// set alarm class
SIf.Alm[1].eAlmClass := E_AlmClass.EOFF;
SIf.Alm[1].strText := 'Communication Error to Line Controller'; 
SIf.Alm[2].eAlmClass := E_AlmClass.EOFF;
SIf.Alm[2].strText := 'Emergency Button pressed';
SIf.Alm[3].eAlmClass := E_AlmClass.INFO;
SIf.Alm[3].strText := 'Communication Error to Line Controller'; 
SIf.Alm[4].eAlmClass := E_AlmClass.INFO;
SIf.Alm[4].strText := 'Line to charge already busy, Job not possible';
SIf.Alm[5].eAlmClass := E_AlmClass.INFO;
SIf.Alm[5].strText := 'False Job Parameter';
SIf.Alm[6].eAlmClass := E_AlmClass.INFO;
SIf.Alm[6].strText := 'Hashtable full, no more input possible';
SIf.Alm[7].eAlmClass := E_AlmClass.INFO;
SIf.Alm[7].strText := 'Data Channel Error Receive Data';
SIf.Alm[8].eAlmClass := E_AlmClass.INFO;
SIf.Alm[8].strText := 'Data Channel Error Send Data';

//*******************************************************************************
// initial values
//*******************************************************************************
// software configuration
CIf.SwCfg.bolExist := TRUE;
CIf.SwCfg.bolSimulation := FALSE;

// Configuration
SIf.Cfg.bolDtChToLine_send := TRUE;

// parmeter
SIf.Par.udiTimeDriveStart_ms := 2000;
SIf.Par.udiTimeDriveStop_ms := 500;
SIf.Par.udiIntervalBufferFilling_ms:= 2000;
END_METHOD

METHOD PROTECTED getCmdState : STRING
VAR_INPUT
	intCmdState: INT;
	bolState: BOOL;
END_VAR
getCmdState := SUPER^.getCmdState(intCmdState:=intCmdState,bolState:=bolState); // get global/base defined cmds/states
IF (getCmdState='') THEN // global not defined get local
	// get string cmd/state string information in runtime
	IF (bolState=FALSE) THEN
		// cmd's
	ELSE
	
	// cmd's
		CASE intCmdState OF
				
			// SUB States
			cSTA_SUB_INITIALIZED:
				getCmdState := 'cSTA_SUB_INITIALIZED';
			cSTA_SUB_START_CYCLE:
				getCmdState := 'cSTA_SUB_START_CYCLE';
			cSTA_SUB_START_Wait_CYCLE:
				getCmdState := 'cSTA_SUB_START_Wait_CYCLE';
			cSTA_SUB_START_ELEMENTS:
				getCmdState := 'cSTA_SUB_START_ELEMENTS';
			cSTA_SUB_START_INLET:
				getCmdState := 'cSTA_SUB_START_INLET';
			cSTA_SUB_START_FINAL:
				getCmdState := 'cSTA_SUB_START_FINAL';
		
			cSTA_SUB_STOP_INLET:
				getCmdState := 'cSTA_SUB_STOP_INLET';
			cSTA_SUB_STOP_CYCLE:
				getCmdState := 'cSTA_SUB_STOP_CYCLE';
			cSTA_SUB_STOP_Wait_CYCLE:
				getCmdState := 'cSTA_SUB_STOP_Wait_CYCLE';
			cSTA_SUB_STOP_ELEMENTS:
				getCmdState := 'cSTA_SUB_STOP_ELEMENTS';
			cSTA_SUB_STOP_OUTLET:
				getCmdState := 'cSTA_SUB_STOPP_OUTLET';
			cSTA_SUB_ERROR:
				getCmdState := 'cSTA_SUB_ERROR';
			cSTA_SUB_FINISHED:
				getCmdState := 'cSTA_SUB_FINISHED';

			cSTA_SUB_RUN_WAIT_JOB:
				getCmdState := 'cSTA_SUB_RUN_WAIT_JOB';
			cSTA_SUB_RUN_SET_PAR:
				getCmdState := 'cSTA_SUB_RUN_SET_PAR';
			cSTA_SUB_RUN_SET_CMD:
				getCmdState := 'cSTA_SUB_RUN_SET_CMD';
			cSTA_SUB_RUN_WAIT_DONE:
				getCmdState := 'cSTA_SUB_RUN_WAIT_DONE';
			cSTA_SUB_RUN_UPDATE:
				getCmdState := 'cSTA_SUB_RUN_UPDATE';

		END_CASE;
	END_IF
END_IF
END_METHOD

METHOD getCtrlSIf : POINTER TO T_Ctrl_SIf_HPS
getCtrlSIf := ADR(SIf);
END_METHOD

METHOD PROTECTED IoInBridge : BOOL
// digitale and analoge inputs read from hardware or forcing
SIf.In.bolCounterIn1.map := THIS^.In_bolCounterIn1;
SIf.In.bolCounterIn2.map := THIS^.In_bolCounterIn2;
SIf.In.bolCounterOut1.map := THIS^.In_bolCounterOut1;
SIf.In.bolCounterOut2.map := THIS^.In_bolCounterOut2;
SIf.In.bolBringShirtStraight .map := THIS^.In_bolBringShirtStraight;
SIf.In.bolBringShirtTurned .map := THIS^.In_bolBringShirtTurned;

IF (CIf.SwCfg.bolSimulation = FALSE) THEN
	getInBol(CIf.Job.bolIoForce,ADR(SIf.In.bolCounterIn1));
	getInBol(CIf.Job.bolIoForce,ADR(SIf.In.bolCounterIn2));
	getInBol(CIf.Job.bolIoForce,ADR(SIf.In.bolCounterOut1));
	getInBol(CIf.Job.bolIoForce,ADR(SIf.In.bolCounterOut2));
	getInBol(CIf.Job.bolIoForce,ADR(SIf.In.bolBringShirtStraight));
	getInBol(CIf.Job.bolIoForce,ADR(SIf.In.bolBringShirtTurned));
ELSE
	//simulation of global IO
END_IF
END_METHOD

METHOD PROTECTED IoOutBridge : BOOL
// digitale and analoge inputs read from hardware or forcing
IF (CIf.SwCfg.bolSimulation = FALSE) THEN
	// check interlocks to prevent damages
	IF (CIf.Job.bolIlkOverwrite=FALSE) THEN
	
		;
	END_IF
	
	// Outputs for Interface to HeatPress without LineControl
	setOutBol(CIf.Job.bolIoForce ,ADR(SIf.Out.bolShirtStraightReady));
	setOutBol(CIf.Job.bolIoForce ,ADR(SIf.Out.bolShirtTurnReady));	
	THIS^.Out_ShirtStraightReady := SIf.Out.bolShirtStraightReady.map;
	THIS^.Out_ShirtTurnReady := SIf.Out.bolShirtTurnReady.map;
	
END_IF
END_METHOD

METHOD RefillTurnedLine
VAR
	/// Loop variable
	ii: INT;
END_VAR
// Simulation
IF (CIf.SwCfg.bolSimulation) THEN
;
END_IF
	
	
// Method refill all zones
CASE SubStateMachineRefill OF		
			
	// Check space in buffer X
	//-------------------------------
	0:
		// Check if number of hangers "per Pulse" have space in the next buffer
		// Condition: (zone[X].NumOfHangers + zone[ X + 1] .NumOfHangersPerPuls) < zone[X].MaxCapacity   			
		IF ((pSEP_SIF^.Cur.dinNumOfHangersInBuffer < pSEP_SIF^.Cfg.dinMaxCapacity) AND 
			(pSLB_T_SIF^.Cur.dinNumOfHangersInBuffer <> 0) AND (pSLB_T_SIF^.Cur.bolHangerDetected = TRUE)) THEN
			
			// Send release command to buffer zone X+1
			pSLB_T_CIF^.Job.intACmd:= SLB_CmdState.cCMD_RELEASE;	
			SubStateMachineRefill:= 1;						
		END_IF
	
	// Check if zone X+1 is released
	//-------------------------------
	1:
		IF(pSLB_T_CIF^.Job.intACmd = BASE_PLC.cCMD_DONE)THEN
			// Send stop command to buffer zone X+1
			SubStateMachineRefill:= 2;
			// Counter correction if no counter at inside of Buffer
			IF pSEP_SIF^.Cfg.bolHasBufferFullSensor = FALSE THEN
				pSEP_SIF^.Cur.dinNumOfHangersInBuffer := pSEP_SIF^.Cur.dinNumOfHangersInBuffer + 1;
			END_IF
		END_IF	
	
	// Check if zone X+1 is stopped
	//-------------------------------
	2:
		udiTimeInStateRefill_ms:= 0;
		SubStateMachineRefill:= 3;
		pHRU_CIF^.Job.intACmd := cCMD_RUN;	// Set Command to HRU				
	
	// Check if HRU is done
	//-------------------------------
	3: 
		IF (pHRU_CIf^.Job.intACmd = cSTA_DONE) THEN							// Hanger Rotation Unit done
			SubStateMachineRefill:= 4;
		END_IF

		
	// Break
	//-------------------------------
	4:	
		// Increment time in state	
		udiTimeInStateRefill_ms:= udiTimeInStateRefill_ms + me.FUBInfo.udiSample_ms;
		IF (udiTimeInStateRefill_ms > SIf.Par.udiIntervalBufferFilling_ms) THEN
			// Back to first state
			SubStateMachineRefill:= 0;	
		END_IF
		
END_CASE
END_METHOD

METHOD PROTECTED sta_OFF : BOOL
// state implemetation
//--------------------------------------------------------------------------------------
// Entry action
	IF (me.StateMachine.intState<>me.StateMachine.intStateLastCycle) THEN
		me.StateMachine.intStateLastCycle := me.StateMachine.intState;
		
	END_IF


//--------------------------------------------------------------------------------------
// Cyclic action
	IF (me.StateMachine.intState=me.StateMachine.intStateLastCycle) THEN
		
		;
		
		
		// State Change Condition
		IF (me.intCmd=cCMD_RUN) THEN
			me.StateMachine.intStateNext :=  cSTA_RUNBusy;
		END_IF
	END_IF




//--------------------------------------------------------------------------------------
// Exit action
	IF (me.StateMachine.intState<>me.StateMachine.intStateNext) THEN
		;
	END_IF
END_METHOD

METHOD PROTECTED sta_RUN : BOOL
// state implemetation
//--------------------------------------------------------------------------------------
// Entry action
	IF (me.StateMachine.intState<>me.StateMachine.intStateLastCycle) THEN
		me.StateMachine.intStateLastCycle := me.StateMachine.intState;
		
		me.SubStateMachine.intState := cSTA_SUB_RUN_WAIT_JOB; // init sub state machine
		me.SubStateMachine.intStateNext := cSTA_SUB_RUN_WAIT_JOB; // init sub state machine

	END_IF


//--------------------------------------------------------------------------------------
// Cyclic action
	IF (me.StateMachine.intState=me.StateMachine.intStateLastCycle) THEN

		// Simulation
		IF (CIf.SwCfg.bolSimulation) THEN
			;
		END_IF

		// Get emptying command from Line with Data Channel
		// Communication to the Line Controll over Data Channel
		THIS^.DtChnToPLC_NewCharge();
		fbDtChnToLine_ChargeDone.bolResetError := CIf.Job.bolAlmReset;
		fbDtChnToLine_ChargeDone.pSIf := ADR(SIf);
		fbDtChnToLine_ChargeDone();
		IF fbDtChnToLine_ChargeDone.intError <> 0 THEN
			// Set Alarm: SIf.Alm[8].strText := 'Data Channel Error Send Data';
			pfbAlarmCtrl^.setAlarm(CIf.Info.intCtrlId,8,fbDtChnToLine_ChargeDone.intError,ADR(SIf.Alm),E_AlmState.RST,CIf.Job.eMe_ActivAlmClass);	
		END_IF
	
		// Start Cycle with substates	
		//--------------------------------------------------------------------------------------
		// sub state machine for sequence
		CASE me.SubStateMachine.intState OF
			//--------------------------------------------------------------------------------------
			
			cSTA_SUB_RUN_WAIT_JOB:
				//--------------------------------------------------------------
				// Job can be set on 3 different ways:
				// 1. Over data channel from Line Controller
				// 2. By digital input (output on heatpress)
				// 3. Over ADS data channel from heatpress
				//--------------------------------------------------------------
				IF ((aTblCharge[0] > 0) 
				OR (SIf.In.bolBringShirtStraight.intern AND NOT bolREBringShirtStraight)
				OR (SIf.In.bolBringShirtTurned.intern AND NOT bolREBringShirtTurned)
				OR (SIf.Ads.stRead.udiRequestBackShirt <> udiRequestBackShirtOld)
				OR (SIf.Ads.stRead.udiRequestFrontShirt <> udiRequestFrontShirtOld)) THEN																	
					me.SubStateMachine.intStateNext := cSTA_SUB_RUN_SET_CMD;
				END_IF
							
				// Interface to HeatPress without LineControl
				SIf.Out.bolShirtStraightReady.intern := pSLB_S_SIF^.Cur.bolHangerDetected; 	// Sensor SEP7 has Hanger detected
				SIf.Out.bolShirtTurnReady.intern := pSEP_SIF^.Cur.bolHangerDetected; // pSLB_T_SIF^.Cur.bolHangerDetected;		// Sensor SEP6 has Hanger detected
				
			cSTA_SUB_RUN_SET_CMD:
				// Digital Input or ADS has priority to the data channel
				// get the correct Common interface to set the RELEASE Command
				IF ((SIf.In.bolBringShirtStraight.intern = TRUE) OR (SIf.Ads.stRead.udiRequestFrontShirt <> udiRequestFrontShirtOld)) THEN
					udiRequestFrontShirtOld:= SIf.Ads.stRead.udiRequestFrontShirt; 
					pSLB_WORK_CIF := pSLB_S_CIF;
				ELSIF ((SIf.In.bolBringShirtTurned.intern = TRUE) OR (SIf.Ads.stRead.udiRequestBackShirt <> udiRequestBackShirtOld)) THEN
					udiRequestBackShirtOld:= SIf.Ads.stRead.udiRequestBackShirt; 
					pSLB_WORK_CIF := pSEP_CIF; //pSLB_T_CIF;	
				ELSIF (aTblCharge[0] = 1) THEN
					// If job from Datachannel, save the line number
					usiLineAct := INT_TO_USINT(aTblCharge[0]);
					pSLB_WORK_CIF := pSLB_S_CIF;
				ELSIF (aTblCharge[0] = 2) THEN
					// If job from Datachannel, save the line number
					usiLineAct := INT_TO_USINT(aTblCharge[0]);
					pSLB_WORK_CIF := pSEP_CIF; //pSLB_T_CIF;
				END_IF
				
				// Send Release command to the correct job interface to release one hanger 
				pSLB_WORK_CIF^.Job.intACmd := STB_CmdState.cCMD_RELEASE;				
(*				// Send Run command to HRU if Shirt is in Turn Line
				IF (pSLB_WORK_CIF^.Info.intCtrlId = pSLB_T_CIF^.Info.intCtrlId) THEN	// Check if Shirt is in Turn Line
					pHRU_CIF^.Job.intACmd := cCMD_RUN;									// Send Command Run to HRU
				END_IF
*)		
				// Interface to HeatPress without LineControl
				SIf.Out.bolShirtStraightReady.intern := FALSE; 	// Not Ready
				SIf.Out.bolShirtTurnReady.intern := FALSE;		// Not Ready
				
				me.SubStateMachine.intStateNext := cSTA_SUB_RUN_WAIT_DONE;
			
			cSTA_SUB_RUN_WAIT_DONE:
				IF (pSLB_WORK_CIF^.Job.intACmd = cSTA_DONE) THEN
					IF (pSLB_WORK_CIF^.Info.intCtrlId = pSEP_CIF^.Info.intCtrlId) THEN		// Check if Shirt is in Turn Line
						pSLB_WORK_CIF^.Job.intACmd := BASE_PLC.cCMD_STOP;
(*						IF (pHRU_CIf^.Job.intACmd = cSTA_DONE) THEN							// Hanger Rotation Unit done
							me.SubStateMachine.intStateNext := cSTA_SUB_RUN_SET_RELEASE;
						ELSIF (pHRU_CIf^.Job.intState = cSTA_ERROR) THEN					// Hanger Rotation Unit failed
							me.SubStateMachine.intStateNext := cSTA_SUB_ERROR;
						END_IF
					ELSE																	// Straight Line -> no HRU check required
*)					END_IF
					me.SubStateMachine.intStateNext := cSTA_SUB_RUN_UPDATE;
				END_IF
				
(*			cSTA_SUB_RUN_SET_RELEASE:		// SEP between HRU and SLS
				IF (pSEP_SIF^.Cur.bolHangerDetected = TRUE) THEN
					pSEP_CIF^.Job.intACmd := STB_CmdState.cCMD_RELEASE;
					me.SubStateMachine.intStateNext := cSTA_SUB_RUN_WAIT_RELEASED;
				END_IF
				
			cSTA_SUB_RUN_WAIT_RELEASED:		// SEP between HRU and SLS
				IF (pSEP_CIF^.Job.intACmd = BASE_PLC.cSTA_DONE) THEN
					me.SubStateMachine.intStateNext := cSTA_SUB_RUN_UPDATE;
					pSEP_CIF^.Job.intACmd := BASE_PLC.cCMD_STOP;
				END_IF
*)				
			cSTA_SUB_RUN_UPDATE:
				// only delete the table if the job was from the table
				IF 	usiLineAct = INT_TO_USINT(aTblCharge[0]) THEN
					FOR intI := 0 TO (cintMaxCharge-1) DO
						aTblCharge[intI] := aTblCharge[intI+1];
					END_FOR
					aTblCharge[cintMaxCharge-1] := 0;
				END_IF
				usiLineAct := 0;
				
				// Send a message over Datachannel to the linecontroler
				IF (SIf.Cfg.bolDtChToLine_send = TRUE) THEN	
					intDtChnToLineState	:= fbDtChnToLine_ChargeDone.Creat(In_intLine := USINT_TO_INT(usiLineAct));
					IF  intDtChnToLineState < 0 THEN
						// SIf.Alm[8].strText := 'Data Channel Error Send Data';
						pfbAlarmCtrl^.setAlarm(CIf.Info.intCtrlId,8,intDtChnToLineState,ADR(SIf.Alm),E_AlmState.RST,CIf.Job.eMe_ActivAlmClass);
					END_IF
				END_IF
				
				me.SubStateMachine.intStateNext := cSTA_SUB_RUN_WAIT_JOB;
				
			cSTA_SUB_ERROR:
				; // Do nothing
					
		END_CASE
		
		//----------------------------------------------------------------------
		// Continuous refill of last SEP
		//----------------------------------------------------------------------
		THIS^.RefillTurnedLine();
		
		// Rising Edge detection of inputs
		bolREBringShirtStraight:= SIf.In.bolBringShirtStraight.intern;
		bolREBringShirtTurned:= SIf.In.bolBringShirtTurned.intern;

		
		me.SubStateMachine.intStateLastCycle := me.SubStateMachine.intState;
		CIf.Job.strSubState := THIS^.getCmdState(intCmdState:=me.SubStateMachine.intState,bolState:=TRUE);
		IF (me.SubStateMachine.intState<>me.SubStateMachine.intStateNext) THEN
			me.SubStateMachine.intState := me.SubStateMachine.intStateNext;  // set next state for next cycle
			me.SubStateMachine.udiTimeInState_ms := 0; // reset timer
			// log state change -> open point
		ELSE
			// increment time in state	
			me.SubStateMachine.udiTimeInState_ms := me.SubStateMachine.udiTimeInState_ms + me.FUBInfo.udiSample_ms;
		END_IF
				
		// State Change Condition	
		IF ((me.intCmd=cCMD_STOP) AND (me.SubStateMachine.intStateNext = cSTA_SUB_RUN_WAIT_JOB)) THEN
			me.StateMachine.intStateNext :=  cSTA_STOPBusy;	
		END_IF
		
		IF ((me.intCmd=cCMD_STOP) AND (me.SubStateMachine.intStateNext = cSTA_SUB_ERROR)) THEN
			me.StateMachine.intStateNext :=  cSTA_STOPBusy;	
		END_IF

	END_IF




//--------------------------------------------------------------------------------------
// Exit action
	IF (me.StateMachine.intState<>me.StateMachine.intStateNext) THEN
		// Interface to HeatPress without LineControl
		SIf.Out.bolShirtStraightReady.intern := FALSE; 	// Not Ready
		SIf.Out.bolShirtTurnReady.intern := FALSE;		// Not Ready
	END_IF
END_METHOD

METHOD PROTECTED sta_RUNBusy : BOOL
// state implemetation
//--------------------------------------------------------------------------------------
// Entry action
	IF (me.StateMachine.intState<>me.StateMachine.intStateLastCycle) THEN
		me.StateMachine.intStateLastCycle := me.StateMachine.intState;
		
		me.SubStateMachine.intState := cSTA_SUB_INITIALIZED; // init sub state machine
		me.SubStateMachine.intStateNext := cSTA_SUB_INITIALIZED; // init sub state machine
		
		fbSimulationTimer.IN := FALSE;
		fbSimulationTimer.PT := UDINT_TO_TIME(SIf.Par.udiTimeOutRead_ms);
		fbSimulationTimer(); // set time/reset timer
		fbSimulationTimer.IN := TRUE; // start timer
	END_IF


//--------------------------------------------------------------------------------------
// Cyclic action
	IF (me.StateMachine.intState=me.StateMachine.intStateLastCycle) THEN

		// Simulation
		IF (CIf.SwCfg.bolSimulation) THEN
			fbSimulationTimer(); // simulation time
			IF (fbSimulationTimer.Q) THEN
				;
			END_IF
		END_IF
		
		// Cyclicle action
		// Start Cycle with substates	
		//--------------------------------------------------------------------------------------
		// sub state machine for sequence
		CASE me.SubStateMachine.intState OF
			//--------------------------------------------------------------------------------------
			cSTA_SUB_INITIALIZED:
				me.SubStateMachine.intStateNext := cSTA_SUB_START_ELEMENTS;
				
			cSTA_SUB_START_ELEMENTS:
				// Start Slidbuffers
				pSLB_S_CIF^.Job.intACmd := cCMD_RUN;
				pSLB_T_CIF^.Job.intACmd := cCMD_RUN;
				// Start Hanger Rotation Unit
				// pHRU_CIF^.Job.intACmd := cCMD_RUN;	// In this state no RUN needed

				IF ((pSLB_S_CIF^.Job.intState = cSTA_RUN) AND (pSLB_T_CIF^.Job.intState = cSTA_RUN)
					 (*AND (pHRU_CIF^.Job.intState = cSTA_RUN)*)) THEN		// is not in RUN
					intDriveIndex := (usiNumOfMultiChild-1);
					me.SubStateMachine.intStateNext := cSTA_SUB_START_CYCLE;
				END_IF
					
			cSTA_SUB_START_CYCLE:
				//start all Buffers and Desicion Points
				a_pMultiChildCIF[intDriveIndex]^.Job.intACmd := cCMD_RUN;
				
				IF a_pMultiChildCIF[intDriveIndex]^.Job.intState = cSTA_RUN THEN
					me.SubStateMachine.intStateNext := cSTA_SUB_START_Wait_CYCLE;
				END_IF
				
			cSTA_SUB_START_Wait_CYCLE:								
				IF (me.SubStateMachine.udiTimeInState_ms >= SIf.Par.udiTimeDriveStart_ms) THEN
					IF intDriveIndex = 0 THEN
						me.SubStateMachine.intStateNext := cSTA_SUB_START_FINAL;
					ELSE
						intDriveIndex := intDriveIndex - 1;
						me.SubStateMachine.intStateNext := cSTA_SUB_START_CYCLE;
					END_IF
				END_IF
				
			cSTA_SUB_START_FINAL:
					me.SubStateMachine.intStateNext := cSTA_SUB_FINISHED;

		//--------------------------------------------------------------------------------------
			cSTA_SUB_FINISHED:
					;
					
		END_CASE
		me.SubStateMachine.intStateLastCycle := me.SubStateMachine.intState;
		CIf.Job.strSubState := THIS^.getCmdState(intCmdState:=me.SubStateMachine.intState,bolState:=TRUE);
		IF (me.SubStateMachine.intState<>me.SubStateMachine.intStateNext) THEN
			me.SubStateMachine.intState := me.SubStateMachine.intStateNext;  // set next state for next cycle
			me.SubStateMachine.udiTimeInState_ms := 0; // reset timer
			// log state change -> open point
		ELSE
			// increment time in state	
			me.SubStateMachine.udiTimeInState_ms := me.SubStateMachine.udiTimeInState_ms + me.FUBInfo.udiSample_ms;
		END_IF
		
		
		// State Change Condition
		IF (me.SubStateMachine.intState = cSTA_SUB_FINISHED) THEN
			me.StateMachine.intStateNext := cSTA_RUN;
		ELSIF (me.intCmd=cCMD_STOP) THEN
			me.StateMachine.intStateNext :=  cSTA_STOPBusy;	
		END_IF
	END_IF




//--------------------------------------------------------------------------------------
// Exit action
	IF (me.StateMachine.intState<>me.StateMachine.intStateNext) THEN
		;
	END_IF
END_METHOD

METHOD PROTECTED sta_STOP : BOOL
// state implemetation
//--------------------------------------------------------------------------------------
// Entry action
	IF (me.StateMachine.intState<>me.StateMachine.intStateLastCycle) THEN
		me.StateMachine.intStateLastCycle := me.StateMachine.intState;
		
	END_IF


//--------------------------------------------------------------------------------------
// Cyclic action
	IF (me.StateMachine.intState=me.StateMachine.intStateLastCycle) THEN
		
		;
		
		
		// State Change Condition
		IF (me.intCmd=cCMD_RUN) THEN
			me.StateMachine.intStateNext :=  cSTA_RUNBusy;
		END_IF
	END_IF




//--------------------------------------------------------------------------------------
// Exit action
	IF (me.StateMachine.intState<>me.StateMachine.intStateNext) THEN
		;
	END_IF
END_METHOD

METHOD PROTECTED sta_STOPBusy : BOOL
// state implemetation
//--------------------------------------------------------------------------------------
// Entry action
	IF (me.StateMachine.intState<>me.StateMachine.intStateLastCycle) THEN
		me.StateMachine.intStateLastCycle := me.StateMachine.intState;
		
		me.SubStateMachine.intState := cSTA_SUB_INITIALIZED; // init sub state machine
		me.SubStateMachine.intStateNext := cSTA_SUB_INITIALIZED; // init sub state machine
		
		fbSimulationTimer.IN := FALSE;
		fbSimulationTimer.PT := UDINT_TO_TIME(SIf.Par.udiTimeOutRead_ms);
		fbSimulationTimer(); // set time/reset timer
		fbSimulationTimer.IN := TRUE; // start timer
	END_IF


//--------------------------------------------------------------------------------------
// Cyclic action
	IF (me.StateMachine.intState=me.StateMachine.intStateLastCycle) THEN

		// Simulation
		IF (CIf.SwCfg.bolSimulation) THEN
			fbSimulationTimer(); // simulation time
			IF (fbSimulationTimer.Q) THEN
				;
			END_IF
		END_IF
		
		// Cyclicle action
		// Stop Cycle with substates	
		//--------------------------------------------------------------------------------------
		// sub state machine for sequence
		CASE me.SubStateMachine.intState OF
			//--------------------------------------------------------------------------------------
			cSTA_SUB_INITIALIZED:
				me.SubStateMachine.intStateNext := cSTA_SUB_STOP_ELEMENTS;
										
			cSTA_SUB_STOP_ELEMENTS: 
				// Stopp Slidebuffers
				pSLB_S_CIF^.Job.intACmd := cCMD_STOP;
				pSLB_T_CIF^.Job.intACmd := cCMD_STOP;
				IF ((pSLB_S_CIF^.Job.intState = cSTA_STOP) AND (pSLB_S_CIF^.Job.intState = cSTA_STOP)) THEN
					me.SubStateMachine.intStateNext := cSTA_SUB_STOP_CYCLE;
					intDriveIndex := 0;
				END_IF

			cSTA_SUB_STOP_CYCLE:
				//start all Buffers and Desicion Points
				a_pMultiChildCIF[intDriveIndex]^.Job.intACmd := cCMD_OFF;
				
				IF a_pMultiChildCIF[intDriveIndex]^.Job.intState = cSTA_OFF THEN
					me.SubStateMachine.intStateNext := cSTA_SUB_STOP_Wait_CYCLE;
				END_IF
				
			cSTA_SUB_STOP_Wait_CYCLE:								
				IF (me.SubStateMachine.udiTimeInState_ms >= SIf.Par.udiTimeDriveStart_ms) THEN
					IF intDriveIndex >= (usiNumOfMultiChild-1) THEN
						me.SubStateMachine.intStateNext := cSTA_SUB_STOP_OUTLET;
					ELSE
						intDriveIndex := intDriveIndex + 1;
						me.SubStateMachine.intStateNext := cSTA_SUB_STOP_CYCLE;
					END_IF
				END_IF
			
			cSTA_SUB_STOP_OUTLET:	
				// Stopp Hanger Rotation Unit
				pHRU_CIF^.Job.intACmd := cCMD_OFF;
				IF (pHRU_CIF^.Job.intState = cSTA_OFF) THEN
					me.SubStateMachine.intStateNext := cSTA_SUB_FINISHED;
				END_IF

		
			
			//--------------------------------------------------------------------------------------
			cSTA_SUB_FINISHED:
					;
					
		END_CASE
		me.SubStateMachine.intStateLastCycle := me.SubStateMachine.intState;
		CIf.Job.strSubState := THIS^.getCmdState(intCmdState:=me.SubStateMachine.intState,bolState:=TRUE);
		IF (me.SubStateMachine.intState<>me.SubStateMachine.intStateNext) THEN
			me.SubStateMachine.intState := me.SubStateMachine.intStateNext;  // set next state for next cycle
			me.SubStateMachine.udiTimeInState_ms := 0; // reset timer
			// log state change -> open point
		ELSE
			// increment time in state	
			me.SubStateMachine.udiTimeInState_ms := me.SubStateMachine.udiTimeInState_ms + me.FUBInfo.udiSample_ms;
		END_IF
		
		
		// State Change Condition
		IF (me.SubStateMachine.intState = cSTA_SUB_FINISHED) THEN
			me.StateMachine.intStateNext := cSTA_STOP;
		ELSIF (me.intCmd=cCMD_RUN) THEN
			me.StateMachine.intStateNext :=  cSTA_RUNBusy;	
		END_IF
	END_IF




//--------------------------------------------------------------------------------------
// Exit action
	IF (me.StateMachine.intState<>me.StateMachine.intStateNext) THEN
		;
	END_IF
END_METHOD

METHOD PROTECTED StateMachine : BOOL
SUPER^.StateMachine();

// main statemachine of base controller
CASE me.StateMachine.intState OF
    cSTA_RUNBusy: 
        THIS^.sta_RUNBusy();
    cSTA_RUN: 
        THIS^.sta_RUN();
    cSTA_STOPBusy: 
        THIS^.sta_STOPBusy();
    cSTA_STOP: 
        THIS^.sta_STOP();
		
END_CASE;
END_METHOD

END_FUNCTION_BLOCK
